TYPE ST_ProductStats :
STRUCT
   averageWeight : REAL;
   minWeight     : REAL;
   maxWeight     : REAL;
   defectiveCount: INT;
END_STRUCT
END_TYPE

(* stored: Version 1.1.0.1, ProductVersion 3.1.4024.16
   DUT ST_ProductStats: Id {34425556-2792-4816-a45e-6d0d1bd400c4} *)
